// TIA Portal V16 export
// export: Created 2022-09-01T13:36:55.1803964Z, ExportSetting WithDefaults, DisplayName Totally Integrated Automation Portal, DisplayVersion V16, DisplayName TIA Portal Version Control Interface, DisplayVersion V16, DisplayName TIA Portal Openness, DisplayVersion V16, DisplayName STEP 7 Professional, DisplayVersion V16, DisplayName STEP 7 Safety, DisplayVersion V16, DisplayName WinCC Advanced, DisplayVersion V16
DATA_BLOCK "Alarmes"   // DB13
{ S7_Optimized_Access := 'TRUE' }
VERSION : 0.1
// stored: AutoNumber true, IsOnlyStoredInLoadMemory false, IsRetainMemResEnabled false, IsWriteProtectedInAS false, MemoryReserve 100
   VAR
      ALARMES_1 : Word;
      ALARMES_2 : Word;
      ALARME_DISPARO : Bool;
      PRESSÃO_MÁX : Bool;
      XV102_NÃO_ABRIU : Bool;
      XV102_NÃO_FECHOU : Bool;
   END_VAR
   VAR RETAIN
      TEMP_ABERT_XV102 : Time;
      TEMP_FECHO_XV102 : Time;
   END_VAR
BEGIN
END_DATA_BLOCK
